// TIA Portal V18 export
FUNCTION "RTDadv" : Void   // FC10015, FBD
{ S7_Optimized_Access := 'TRUE' }
VERSION : 0.1
// stored: AutoNumber false, IsIECCheckEnabled false, SetENOAutomatically false, UDAEnableTagReadback false
   VAR_INPUT
      iInput : Int;
      rFilterValue : Real;
      rCalibration : Real;
      rDiv : Real;
   END_VAR
   VAR_OUTPUT
      rOutput : Real;
   END_VAR
   VAR_TEMP
      rTemp : Real;
   END_VAR
   VAR CONSTANT
      rMin : Real := -50.0;
      rMax : Real := 150.0;
   END_VAR
BEGIN

REGION Network 1 (SCL)
   #rTemp := INT_TO_REAL(#iInput);
END_REGION

REGION Network 2 (SCL)
   #rTemp := #rTemp / #rDiv;
END_REGION

REGION Network 3 (SCL)
   #rTemp := #rTemp + #rCalibration;
END_REGION

REGION Network 4 (SCL): Filter
END_REGION

REGION Network 5 (SCL): Output
   //xValid := xDiagOK AND (rTempCalc > -250.0) AND (rTempCalc < 1000.0);
   //IF xValid THEN
   //    rTempC := rTempCalc;
   //END_IF;
   //
   #rOutput := #rTemp;
END_REGION
END_FUNCTION
